Fanuc KAREL source: kt00538.KL

-- PROVISIONAL review KL for V940-1; original PC SHA256 8c28384180fefd87d7ccdda20d17c35b8b2f335f9c393e625e21b7f63d631b05
-- Incomplete behavior may be omitted. Consult companion uncertainty JSON. Do not deploy.
PROGRAM KT00538
%NOLOCKGROUP
VAR
  OUT : BOOLEAN
-- UNRESOLVED_DECL P1 type=000199
-- UNRESOLVED_DECL P2 type=000102
BEGIN
  -- V9_ZERO_TABLE_METADATA_HINT layout=0001; no indexed target words; source/name/runtime held
  -- UNRESOLVED_PC offsets 5-20; opcodes 2E,22,32,35
  -- UNRESOLVED_PC offsets 25-58; opcodes 49,7E,49,7E,AC,23
  -- UNRESOLVED_PC offsets 63-67; opcodes 7F
END KT00538
